FUNCTION Convert_UDINT_TO_LREAL : Hresult
VAR_INPUT
	in : UDINT;
	out : REFERENCE TO LREAL;
END_VAR
VAR
	converted : LREAL;
END_VAR
VAR CONSTANT
	INCOMPATIBLE : HRESULT := 16#9811070E;
END_VAR

converted := UDINT_TO_LREAL(in);

IF (LREAL_TO_UDINT(converted) <> in) THEN
	Convert_UDINT_TO_LREAL := INCOMPATIBLE;
	RETURN;
END_IF

out := converted;

END_FUNCTION

(* stored: Version 1.1.0.1, ProductVersion 3.1.4024.12
   POU Convert_UDINT_TO_LREAL: Id {3c02f3fa-7309-4d32-a936-2ed6fcfc0e56}, SpecialFunc None *)
